FUNCTION_BLOCK "Novus_tht"
{ S7_Optimized_Access := 'TRUE' }
VERSION : 0.1
   VAR_INPUT
      mb_addr : USInt;
   END_VAR

   VAR_OUTPUT
      temperature : Int;
      humidity : Int;
   END_VAR

   VAR_IN_OUT
      mb_query : "mb_query";
   END_VAR

   VAR
      s : "mb_station_udt";
      serial_number : DWord;
      raw_values { ExternalAccessible := 'False'; ExternalVisible := 'False'; ExternalWritable := 'False'} : Struct
         temp { ExternalAccessible := 'False'; ExternalVisible := 'False'; ExternalWritable := 'False'} : Int;
         hum { ExternalAccessible := 'False'; ExternalVisible := 'False'; ExternalWritable := 'False'} : Int;
      END_STRUCT;
   END_VAR


BEGIN
	// - Novus - RHT (Temperature transmitter)
	// - http://www.novusautomation.com/downloads/Arquivos/v10x_b_manual_rht_wm-dm-p10_485_lcd_%20english.pdf

	"mb_station_header"(station := #s, mb_query := #mb_query);
	#mb_query.mb_addr := #mb_addr;

	#mb_query.mode := #mb_query.c.read.holding_reg;
	#mb_query(data_addr := 7, data_ptr := #raw_values);
	#mb_query(data_addr := 0, data_ptr := #serial_number);

	"mb_station_footer"(station := #s, mb_query := #mb_query);

	IF #s.out.error_comm THEN
	    #raw_values.temp := 0;
	    #raw_values.hum := 0;
	END_IF;

	#temperature := #raw_values.temp / 10;
	#humidity := #raw_values.hum / 10;

END_FUNCTION_BLOCK

